PROGRAM PRG_11_AirFlowAnalytics
VAR
	AirFlowRateSensor: GenericSensor;
	AirPressureSensor: GenericSensor;
	AirTemperatureSensor: GenericSensor;
	
	{attribute 'OPC.UA.DA' := '0'}
	{attribute 'OPC.UA.DA.Access' := '1'}			// read only
	{attribute 'OPC.UA.DA.StructuredType' := '1'}
	AirFlowRateSensorStruct						: SingleSensor_DataModel;
	
	{attribute 'OPC.UA.DA' := '0'}
	{attribute 'OPC.UA.DA.Access' := '1'}			// read only
	{attribute 'OPC.UA.DA.StructuredType' := '1'}
	AirPressureSensorStruct						: SingleSensor_DataModel;
	
	{attribute 'OPC.UA.DA' := '0'}
	{attribute 'OPC.UA.DA.Access' := '1'}			// read only
	{attribute 'OPC.UA.DA.StructuredType' := '1'}
	AirTemperatureSensorSensorStruct			: SingleSensor_DataModel;
END_VAR

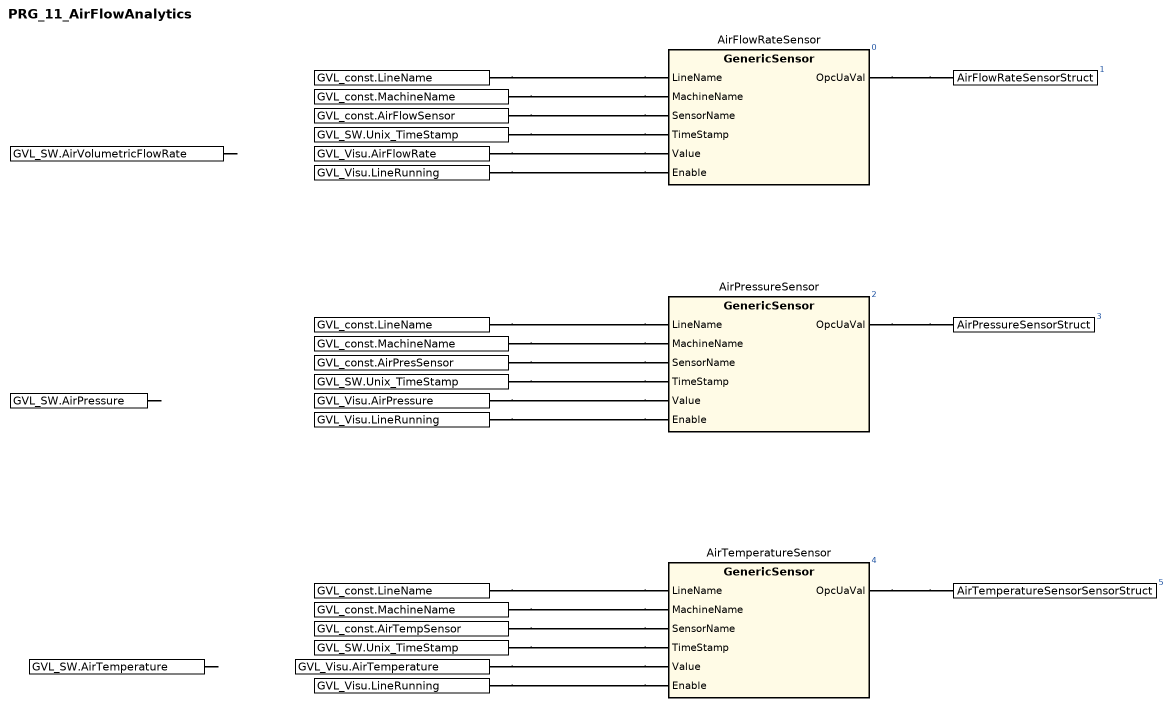
AirFlowRateSensor(
    LineName := GVL_const.LineName,
    MachineName := GVL_const.MachineName,
    SensorName := GVL_const.AirFlowSensor,
    TimeStamp := GVL_SW.Unix_TimeStamp,
    Value := GVL_Visu.AirFlowRate,
    Enable := GVL_Visu.LineRunning); // GenericSensor
AirFlowRateSensorStruct := AirFlowRateSensor.OpcUaVal;
AirPressureSensor(
    LineName := GVL_const.LineName,
    MachineName := GVL_const.MachineName,
    SensorName := GVL_const.AirPresSensor,
    TimeStamp := GVL_SW.Unix_TimeStamp,
    Value := GVL_Visu.AirPressure,
    Enable := GVL_Visu.LineRunning); // GenericSensor
AirPressureSensorStruct := AirPressureSensor.OpcUaVal;
AirTemperatureSensor(
    LineName := GVL_const.LineName,
    MachineName := GVL_const.MachineName,
    SensorName := GVL_const.AirTempSensor,
    TimeStamp := GVL_SW.Unix_TimeStamp,
    Value := GVL_Visu.AirTemperature,
    Enable := GVL_Visu.LineRunning); // GenericSensor
AirTemperatureSensorSensorStruct := AirTemperatureSensor.OpcUaVal;
// GVL_SW.AirVolumetricFlowRate: input not connected
// GVL_SW.AirPressure: input not connected
// GVL_SW.AirTemperature: input not connected

END_PROGRAM

(* stored: Version 1.1.0.1, ProductVersion 3.1.4024.15
   POU PRG_11_AirFlowAnalytics: Id {96d35d53-1242-4be7-b36c-7cd64f603641}, SpecialFunc None *)
